// Mitsubishi GX Works2 project: 31   PLC: FX3G

// task Task_01 (event TRUE, interval 0, priority 31): POU_01

PROGRAM POU_01
VAR
  wstep : INT;
  pwd : INT;
  inPwd : INT;
  money : INT;
  show : INT;
  userInput : INT;
  ton1 : TON;
END_VAR
M99 := FALSE AND
M0 AND M1 AND M2
AND M3 AND M4 AND
Y0 AND Y1;

IF M8002 THEN
    wstep := 0;
    money := 5200;
    pwd := 1234;
END_IF;

IF (wstep <> 0) THEN
	D1 := 0;
END_IF;
IF (wstep <> 60) AND (wstep <> 40)  AND (wstep <> 20)  THEN
	show := -1;
END_IF;
IF (wstep <> 40)  AND (wstep <> 20) THEN
	D3 := -1;
END_IF;

D0:= pwd;
inPwd := D1;
D2 := show;
userInput := D3;

CASE wstep OF
    0:
        Y0 := FALSE;
        Y1 := FALSE;
        IF M0 THEN
            IF (inPwd = pwd) THEN
                wstep := 1;
            ELSE
                wstep  := 2;
  			END_IF;
        END_IF;
    1:
        Y0 := TRUE;

        IF M4 THEN
            wstep := 0;
        ELSIF M1 THEN
            wstep := 20;
        ELSIF M2 THEN
            wstep := 40;
        ELSIF M3 THEN
            wstep := 60;
        END_IF;
    2:
        Y1 := TRUE;
        ton1(in := NOT ton1.q, pt := t#1s);

        IF ton1.q THEN
            wstep := 0;
        END_IF;

    20:
    	show := money;
    	
        IF M0 THEN
            money := money + userInput;
            wstep := 1;
        END_IF;

    40:
    	show := money;
    	
        IF M0 AND (money - userInput >= 0) THEN
            money := money - userInput;
            wstep := 1;
        END_IF;

    60:
        show := money;

        IF M0 THEN
            wstep := 1;
        END_IF;
END_CASE;
END_PROGRAM
